FUNCTION_BLOCK MotorManagement
VAR_IN_OUT
	Motor	: stMotor;
END_VAR

VAR_INPUT
	xIn_StatusDispatch: BOOL;
	xIn_StatusError		: BOOL;
	xIn_StatusRunning	: BOOL;
	xIn_ResetError		: BOOL;
	xIn_AuxPower		: BOOL;
	UseReverse			: BOOL;
	TestMode			: BOOL;
	TriggerForward		: BOOL;
	TriggerReverse		: BOOL;
	TriggerOutsideForTestManualForward: BOOL;
	TriggerOutsideForTestManualReverse: BOOL;
END_VAR
VAR_OUTPUT
	Error	: BOOL;
	ErrorID	: UINT;
END_VAR
VAR
	StatusError			: BOOL;
	MotorCannotRunning	: BOOL;
	PowerOff			: BOOL;
	Timer				: TON;
	LocalSwitch_Off		: BOOL;
END_VAR
VAR // added by the converter: edge detectors and wires of the graphical bodies
    _w1 : BOOL;
END_VAR

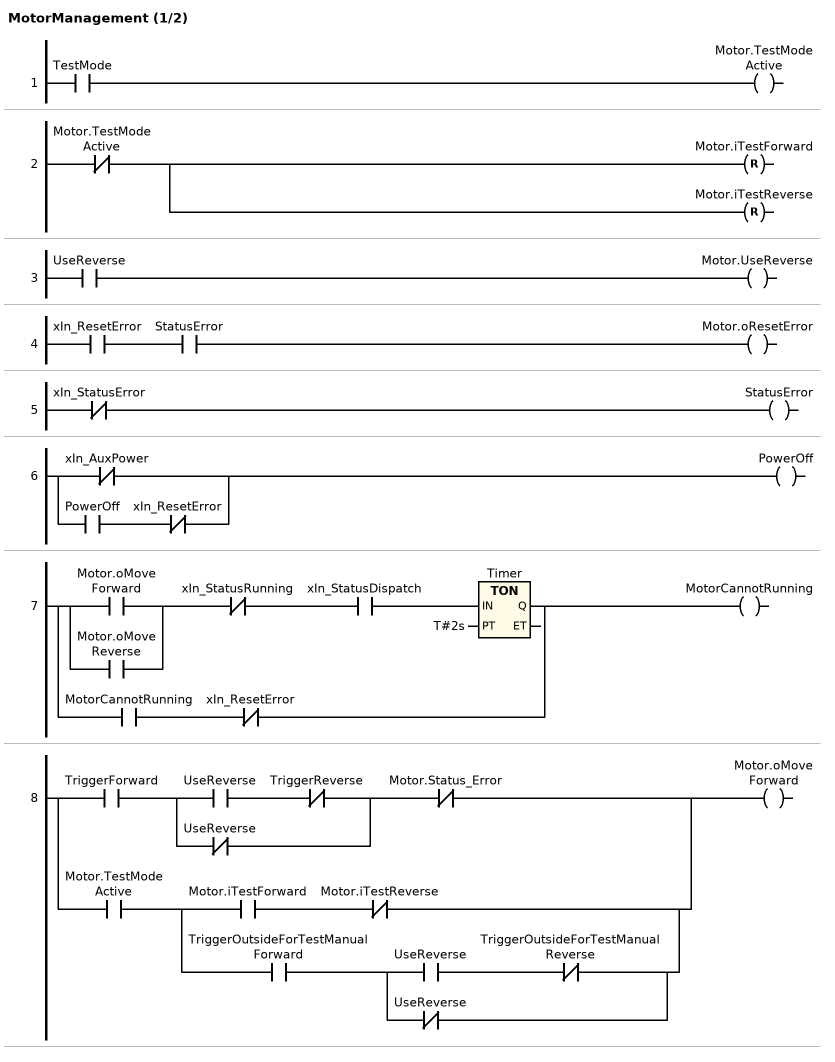
// NETWORK 1
Motor.TestModeActive := TestMode;

// NETWORK 2
_w1 := NOT Motor.TestModeActive;
Motor.iTestForward R= _w1;
Motor.iTestReverse R= _w1;

// NETWORK 3
Motor.UseReverse := UseReverse;

// NETWORK 4
Motor.oResetError := xIn_ResetError AND StatusError;

// NETWORK 5
StatusError := NOT xIn_StatusError;

// NETWORK 6
PowerOff := NOT xIn_AuxPower OR PowerOff AND NOT xIn_ResetError;

// NETWORK 7
Timer(IN := (Motor.oMoveForward OR Motor.oMoveReverse) AND NOT xIn_StatusRunning AND xIn_StatusDispatch, PT := T#2s); // TON
MotorCannotRunning := Timer.Q OR MotorCannotRunning AND NOT xIn_ResetError;

// NETWORK 8
Motor.oMoveForward := TriggerForward AND (UseReverse AND NOT TriggerReverse OR NOT UseReverse) AND NOT Motor.Status_Error OR Motor.TestModeActive AND (Motor.iTestForward AND NOT Motor.iTestReverse OR TriggerOutsideForTestManualForward AND (UseReverse AND NOT TriggerOutsideForTestManualReverse OR NOT UseReverse));

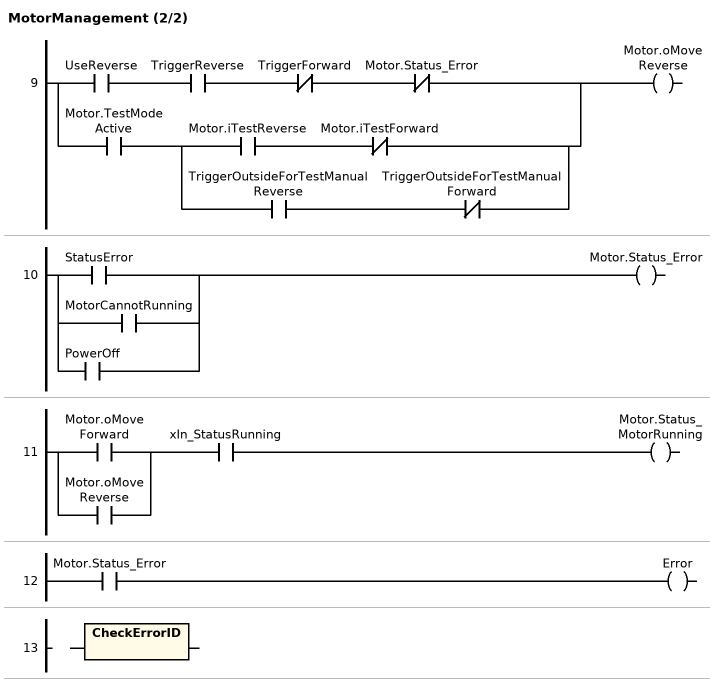
// NETWORK 9
Motor.oMoveReverse := UseReverse AND TriggerReverse AND NOT TriggerForward AND NOT Motor.Status_Error OR Motor.TestModeActive AND (Motor.iTestReverse AND NOT Motor.iTestForward OR TriggerOutsideForTestManualReverse AND NOT TriggerOutsideForTestManualForward);

// NETWORK 10
Motor.Status_Error := StatusError OR MotorCannotRunning OR PowerOff;

// NETWORK 11
Motor.Status_MotorRunning := (Motor.oMoveForward OR Motor.oMoveReverse) AND xIn_StatusRunning;

// NETWORK 12
Error := Motor.Status_Error;

// NETWORK 13
CheckErrorID();

ACTION CheckErrorID:
IF Error THEN
	IF StatusError THEN
		ErrorID:=1;
	ELSIF PowerOff THEN
			ErrorID:=2;
		ELSIF LocalSwitch_Off THEN
				ErrorID:=3;
			ELSIF MotorCannotRunning THEN
					ErrorID:=10;
				ELSE
					ErrorID:=90;
			END_IF
ELSE
	ErrorID:=0;
END_IF

Motor.ErrorID:=ErrorID;
END_ACTION

END_FUNCTION_BLOCK

(* stored: Version 1.1.0.1, ProductVersion 3.1.4024.12
   POU MotorManagement: Id {0fefcc09-5fd1-44ff-a436-967d56300998}, SpecialFunc None
   Action CheckErrorID: Id {ae25c597-c220-4b95-8044-b84b882f4132} *)
